// TIA Portal V19 export
TYPE "LEXCHANGETRAY_typeLogistics_toRollerReq"
// stored: Access Published
   STRUCT
      outFeedReq : Bool;   // 请求排料排料
      inFeedReq : Bool;
   END_STRUCT;
END_TYPE
